TYPE stHMI_COMM :
STRUCT
	_CommunicationConnected : BOOL;
END_STRUCT
END_TYPE

(* stored: Version 1.1.0.1, ProductVersion 3.1.4026.18
   DUT stHMI_COMM: Id {e1786145-24f0-4674-9a44-50c2d5e718ad} *)
